{attribute 'linkalways'} 
{attribute 'no_explicit_call' := 'This FB is a CLASS and must be accessed using methods or properties'}
{attribute 'enable_dynamic_creation'}
FUNCTION_BLOCK _ETcVnFeatureScalingType EXTENDS EnumDatatypeBase
VAR
	localData : ETcVnFeatureScalingType;
	activeData : REFERENCE TO ETcVnFeatureScalingType;
	enumBaseDatatype : _DINT(localData);
END_VAR

METHOD PRIVATE AddLocalEnumeration
VAR_INPUT
	Enumeration : T_MAXSTRING;
	Value : ETcVnFeatureScalingType;
END_VAR
AddEnumeration(Enumeration, Value);
END_METHOD

PROPERTY PUBLIC Address : PVOID
GET
Address := ADR(activeData);
END_GET
END_PROPERTY

METHOD PUBLIC ClearReference
VAR_INPUT
END_VAR
activeData REF= localData;
SetBaseDatatypeReference();
END_METHOD

METHOD PUBLIC Clone : I_Datatype
VAR
    pClone : POINTER TO _ETcVnFeatureScalingType;
END_VAR
pClone := __NEW(_ETcVnFeatureScalingType(InitialValue := Value));
Clone := pClone^;
END_METHOD

METHOD FB_init : BOOL
VAR_INPUT
	bInitRetains : BOOL; // if TRUE, the retain variables are initialized (warm start / cold start)
	bInCopyCode : BOOL;  // if TRUE, the instance afterwards gets moved into the copy code (online change)
	InitialValue : ETcVnFeatureScalingType;
END_VAR
localData := InitialValue;
AddBaseDatatype(enumBaseDatatype);
ClearReference();

AddLocalEnumeration('TCVN_FST1_MAXABS', ETcVnFeatureScalingType.TCVN_FST1_MAXABS);
AddLocalEnumeration('TCVN_FST1_MINMAX', ETcVnFeatureScalingType.TCVN_FST1_MINMAX);
AddLocalEnumeration('TCVN_FST1_STANDARDIZATION', ETcVnFeatureScalingType.TCVN_FST1_STANDARDIZATION);
END_METHOD

PROPERTY PUBLIC Identifier : T_MAXSTRING
GET
Identifier := 'ETcVnFeatureScalingType';
END_GET
END_PROPERTY

METHOD IsEnumeratorValueEqual : BOOL
VAR_INPUT
	Enumerator : I_KeyValueForwardEnumerator;
END_VAR
VAR
	storedValue : ETcVnFeatureScalingType;
END_VAR
IF NOT Enumerator.TryGet(storedValue) THEN
	RETURN;
END_IF

IsEnumeratorValueEqual := storedValue = activeData;
END_METHOD

METHOD PUBLIC MakeReferenceTo
VAR_INPUT
	ReferenceTarget : REFERENCE TO ETcVnFeatureScalingType;
END_VAR
activeData REF= ReferenceTarget;
SetBaseDatatypeReference();
END_METHOD

METHOD PROTECTED SetBaseDatatypeReference
VAR_INPUT
END_VAR
enumBaseDatatype.MakeReferenceTo(activeData);
END_METHOD

PROPERTY PUBLIC Size : UDINT
GET
Size := SIZEOF(activeData);
END_GET
END_PROPERTY

METHOD TryMakeReferenceTo : BOOL
VAR_INPUT
	Target : I_Datatype;
END_VAR
VAR
	targetAsEnum : I_EnumDatatype;
	pTargetData : POINTER TO ETcVnFeatureScalingType;
END_VAR
IF NOT Target.TryResolveAsEnumDatatype(targetAsEnum) THEN
	RETURN;
END_IF

IF targetAsEnum.Identifier <> Identifier THEN
	RETURN;
END_IF

pTargetData := Target.Address;
activeData REF= pTargetData^;
SetBaseDatatypeReference();
TryMakeReferenceTo := TRUE;
END_METHOD

PROPERTY PUBLIC Value : ETcVnFeatureScalingType
GET
Value := activeData;
END_GET
SET
activeData := Value;
END_SET
END_PROPERTY

END_FUNCTION_BLOCK

(* stored: Version 1.1.0.1, ProductVersion 3.1.4024.12
   POU _ETcVnFeatureScalingType: Id {70df1f6e-2a36-017f-1bc4-2c20cd0149af}, SpecialFunc None
   Folder Constructor: Id {7c7f56e0-3589-0463-1832-a3ba2b10ea53}
   Folder Private: Id {a008303e-281a-0f78-1b46-c83332f2a1de}
   Folder Protected: Id {c193fc5d-06ff-0680-2ef4-e79d03c4ca6b}
   Method AddLocalEnumeration: Id {19e1ad55-76bd-0e39-2cfa-65febeb0e046}
   Property Address: Id {6b38cbbc-92e3-0ae2-3964-0362ee5fd100}
   Get Get: Id {be45d830-9b80-0f99-0559-abfd6b4ed908}
   Method ClearReference: Id {b94dfac0-64b6-092f-1934-8145a0ff84c3}
   Method Clone: Id {da488b4d-ee97-067a-2f5c-88c425dbb580}
   Method FB_init: Id {1176f4c8-73a8-06ed-042b-8c10a9cdf229}
   Property Identifier: Id {1c272d41-6da9-0be9-19f1-0c77f1cc7cb4}
   Get Get: Id {34932923-30e8-045b-151f-be7bbfa5c558}
   Method IsEnumeratorValueEqual: Id {a872ee1c-cecf-0500-2607-367a434616ab}
   Method MakeReferenceTo: Id {ec761a61-10c0-0342-11bd-fdae5f816e60}
   Method SetBaseDatatypeReference: Id {29d172cc-9c29-07c9-0635-e80e085d5212}
   Property Size: Id {486f03d9-d2cf-051e-1a4d-84688507073b}
   Get Get: Id {5360a07e-5942-06a3-15d2-2f73aa8b4559}
   Method TryMakeReferenceTo: Id {7611decf-f17c-0cb1-23d6-766ee793c6a5}
   Property Value: Id {b076bf71-76d1-012a-2ec5-d9e3c2e1191f}
   Get Get: Id {2dae3009-0426-0bf3-0aff-7d97d938fcfc}
   Set Set: Id {1ca49788-4eb6-051d-1e4d-65623605610e} *)
